{attribute 'GeneratedUsingTerminal: EP8309-0022-0021'}
{attribute addProperty BoxType "EP8309-0022-0021"}
{attribute addProperty Id "StatusAT %I*Status_6CCA259F6Rotational_SpeedAT %I*INT2Rotation_DirectionAT %I*UINT2"}
{attribute addProperty CRC "3274820158"}
{attribute addProperty Size "10"}
TYPE TACHO_Single_Shaft_Mode_Input_Channel_C331CA3E :
STRUCT
	{attribute addProperty Name "Status"}
	Status AT %I* : Status_6CCA259F;
	{attribute addProperty Name "Rotational_Speed"}
	Rotational_Speed AT %I* : INT;
	{attribute addProperty Name "Rotation_Direction"}
	Rotation_Direction AT %I* : UINT;
END_STRUCT
END_TYPE

(* stored: Version 1.2.0.0, ProductVersion 3.1.4024.9
   DUT TACHO_Single_Shaft_Mode_Input_Channel_C331CA3E: Id {14ef705f-e6bf-4767-a647-6bcf8f5de11c} *)
